{attribute 'qualified_only'}
{attribute 'strict'}
TYPE Test_Enum :
(
	enum_member := 0
);
END_TYPE

(* stored: Version 1.1.0.1, ProductVersion 3.1.4024.13
   DUT Test_Enum: Id {fe5765a6-b39c-4d57-bd06-ebb6324f3917} *)
